VAR_GLOBAL
    bInDeventer : BOOL := FALSE;      // Reiziger is in Deventer
    bKoffieGereed : BOOL := FALSE;    // Koffie is gehaald door koffietaak
    sStatusTekst : STRING := '';      // Status voor visualisatie
END_VAR

(* stored: Version 1.1.0.1, ProductVersion 3.1.4024.15
   GVL GVL: Id {8d0e06c1-69c7-4dc4-8b0b-fcc98f66b25d} *)
